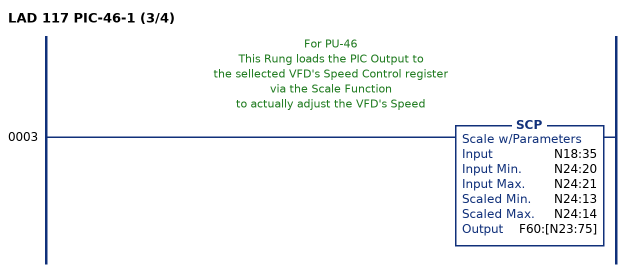
% Rung: 3 %
% For PU-46
% This Rung loads the PIC Output to
% the sellected VFD's Speed Control register
% via the Scale Function
% to actually adjust the VFD's Speed %
SOR SCP N18:35 N24:20 N24:21 N24:13 N24:14 F60:[N23:75] EOR
%   N18:35  PIC461_OUT1  "PIC-46-1 Flash Evap Feed Pres PID Output Value" %
%   N24:20  PID_MIN  "PID Statement Minimum Value" %
%   N24:21  PID_MAX  "PID Statement Maximum Value" %
%   N24:13  AO_MIN_OE4  "Analog Output Minimum Value Generates 4 mA DC (To OE4 AO Module)" %
%   N24:14  AO_MAX_OE4  "Analog Output Maximum Value Generates 20 mA DC (To OE4 AO Module)" %
%   N23:75  PIC461_OUT_PTR  "PIC-46-1 Flash Evap Feed Pres Output Pointer Determines which VFD is controled by FIC" %

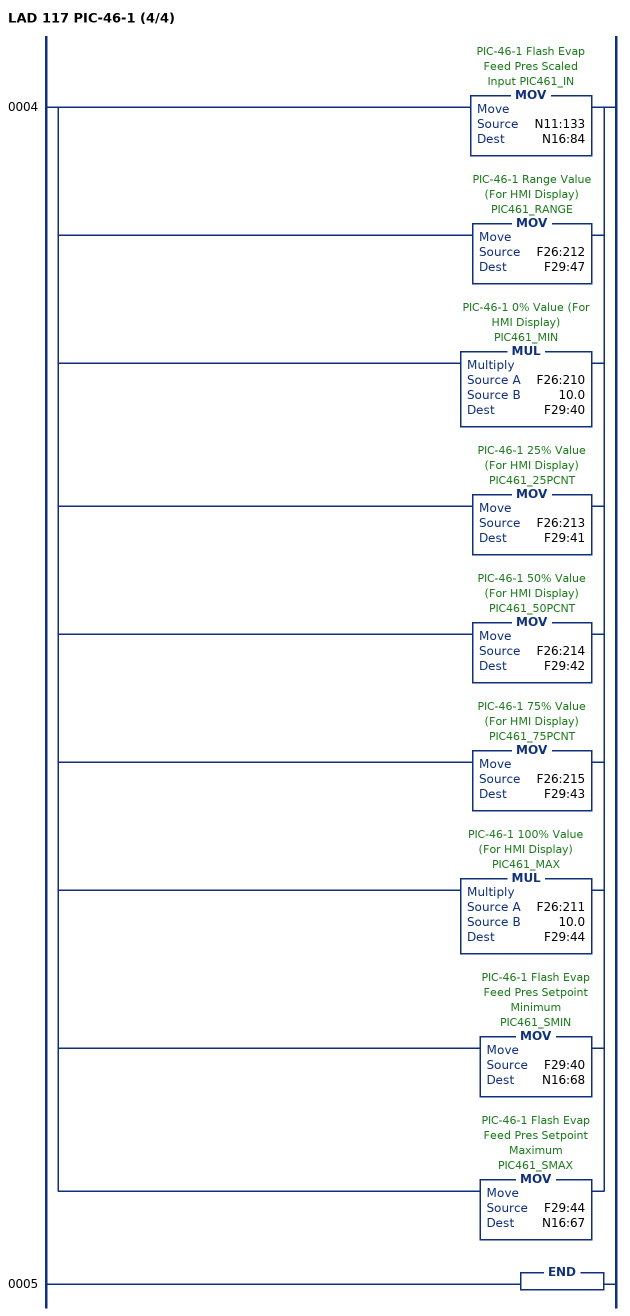
% Rung: 4 %
SOR BST MOV N11:133 N16:84 NXB MOV F26:212 F29:47 NXB MUL F26:210 10.0 F29:40 NXB MOV F26:213 F29:41 NXB MOV F26:214 F29:42 NXB MOV F26:215 F29:43 NXB MUL F26:211 10.0 F29:44 NXB MOV F29:40 N16:68 NXB MOV F29:44 N16:67 BND EOR
%   N11:133  PT461_PID_IN  "PT-46-1 Flash Evap Feed Pres PID Statement Input Value" %
%   N16:84  PIC461_IN  "PIC-46-1 Flash Evap Feed Pres Scaled Input" %
%   F26:212  PT461_RANGE  "PT-46-1 Range Value #NAME?" %
%   F29:47  PIC461_RANGE  "PIC-46-1 Range Value (For HMI Display)" %
%   F26:210  PT461_MIN  "PT-46-1 Minimum Value" %
%   F29:40  PIC461_MIN  "PIC-46-1 0% Value (For HMI Display)" %
%   F26:213  PT461_25PCNT_VALUE  "PT-46-1 25% Range Value For HMI Display" %
%   F29:41  PIC461_25PCNT  "PIC-46-1 25% Value (For HMI Display)" %
%   F26:214  PT461_50PCNT_VALUE  "PT-46-1 50% Range Value For HMI Display" %
%   F29:42  PIC461_50PCNT  "PIC-46-1 50% Value (For HMI Display)" %
%   F26:215  PT461_75PCNT_VALUE  "PT-46-1 75% Range Value For HMI Display" %
%   F29:43  PIC461_75PCNT  "PIC-46-1 75% Value (For HMI Display)" %
%   F26:211  PT461_MAX  "PT-46-1 Maximum Value" %
%   F29:44  PIC461_MAX  "PIC-46-1 100% Value (For HMI Display)" %
%   N16:68  PIC461_SMIN  "PIC-46-1 Flash Evap Feed Pres Setpoint Minimum" %
%   N16:67  PIC461_SMAX  "PIC-46-1 Flash Evap Feed Pres Setpoint Maximum" %
% Rung: 5 %
SOR END EOR

LADDER 121 "TIC-11-1"    % Tempered Water Loop No-1 Temperature PID Controls %
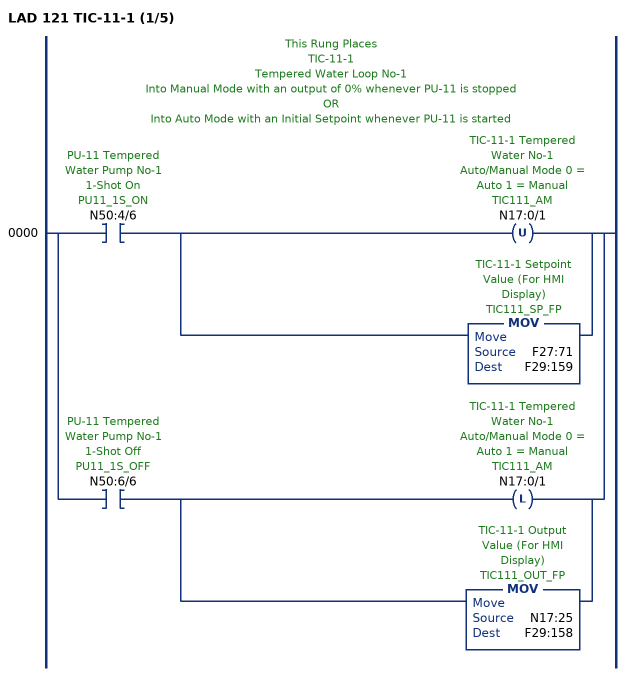
% Rung: 0 %
% This Rung Places
% TIC-11-1
% Tempered Water Loop No-1
% Into Manual Mode with an output of 0% whenever PU-11 is stopped
% OR
% Into Auto Mode with an Initial Setpoint whenever PU-11 is started %
SOR BST XIC N50:4/6 BST OTU N17:0/1 NXB MOV F27:71 F29:159 BND NXB XIC N50:6/6 BST OTL N17:0/1 NXB MOV N17:25 F29:158 BND BND EOR
%   N50:4/6  PU11_1S_ON  "PU-11 Tempered Water Pump No-1 1-Shot On" %
%   N17:0/1  TIC111_AM  "TIC-11-1 Tempered Water No-1 Auto/Manual Mode 0 = Auto 1 = Manual" %
%   F27:71  TIC111_INIT_SP  "TIC-11-1 Initial Temperature Setpoint" %
%   F29:159  TIC111_SP_FP  "TIC-11-1 Setpoint Value (For HMI Display)" %
%   N50:6/6  PU11_1S_OFF  "PU-11 Tempered Water Pump No-1 1-Shot Off" %
%   N17:25  TIC111_OFF_OUTPUT  "TIC-11-1 Output When PU-11 Is Off" %
%   F29:158  TIC111_OUT_FP  "TIC-11-1 Output Value (For HMI Display)" %

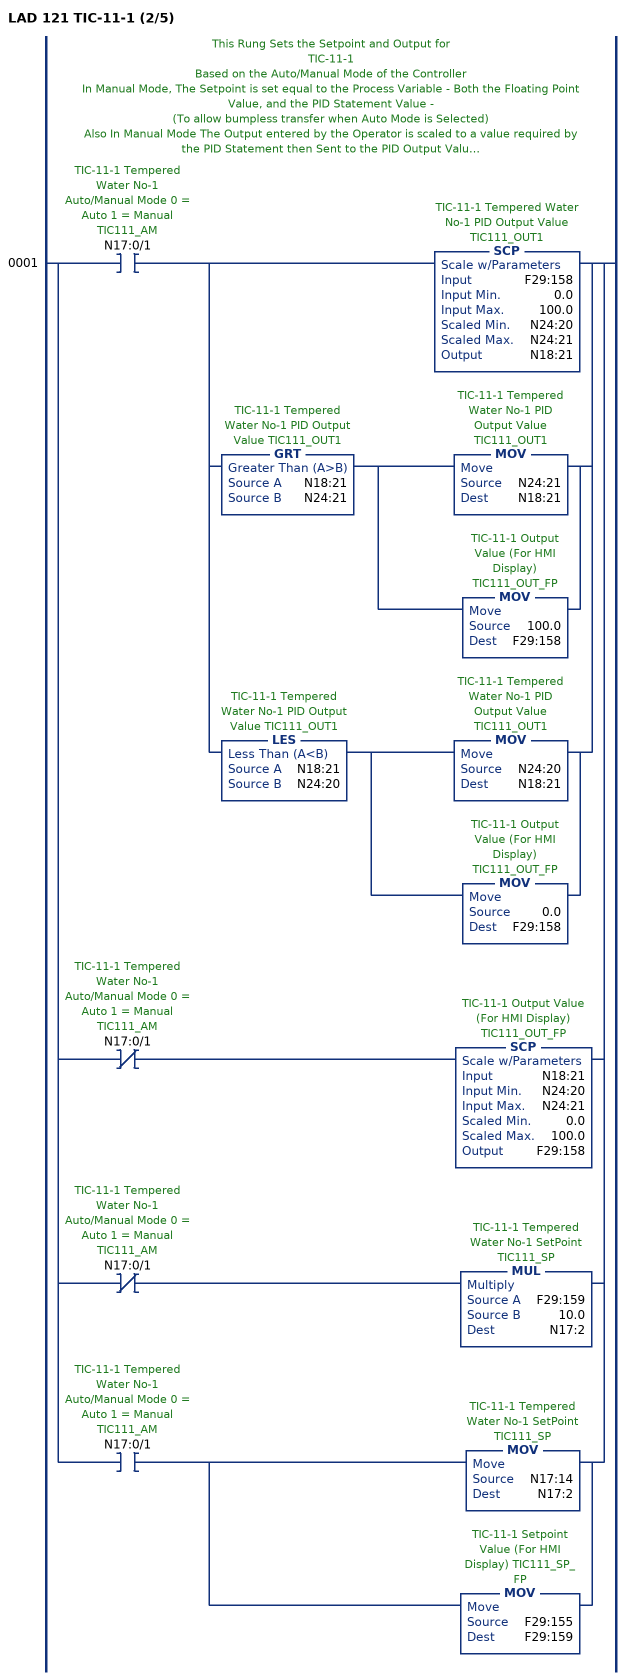
% Rung: 1 %
% This Rung Sets the Setpoint and Output for
% TIC-11-1
% Based on the Auto/Manual Mode of the Controller
% In Manual Mode, The Setpoint is set equal to the Process Variable - Both the Floating Point Value, and the PID Statement Value -
% (To allow bumpless transfer when Auto Mode is Selected)
% Also In Manual Mode The Output entered by the Operator is scaled to a value required by the PID Statement then Sent to the PID Output Value
% 
% In Auto Mode, The Setpoint is Entered by the Operator from Any HMI terminal, Multiplied by 10, and placed in the PID Statement's Setpoint Location
% Also In Auto Mode, the Output (used by the Operator) is set equal to the actual value of the pID statement
% (To allow bumpless transfer when Manual Mode is Selected) %
SOR BST XIC N17:0/1 BST SCP F29:158 0.0 100.0 N24:20 N24:21 N18:21 NXB GRT N18:21 N24:21 BST MOV N24:21 N18:21 NXB MOV 100.0 F29:158 BND NXB LES N18:21 N24:20 BST MOV N24:20 N18:21 NXB MOV 0.0 F29:158 BND BND NXB XIO N17:0/1 SCP N18:21 N24:20 N24:21 0.0 100.0 F29:158 NXB XIO N17:0/1 MUL F29:159 10.0 N17:2 NXB XIC N17:0/1 BST MOV N17:14 N17:2 NXB MOV F29:155 F29:159 BND BND EOR
%   N17:0/1  TIC111_AM  "TIC-11-1 Tempered Water No-1 Auto/Manual Mode 0 = Auto 1 = Manual" %
%   F29:158  TIC111_OUT_FP  "TIC-11-1 Output Value (For HMI Display)" %
%   N24:20  PID_MIN  "PID Statement Minimum Value" %
%   N24:21  PID_MAX  "PID Statement Maximum Value" %
%   N18:21  TIC111_OUT1  "TIC-11-1 Tempered Water No-1 PID Output Value" %
%   F29:159  TIC111_SP_FP  "TIC-11-1 Setpoint Value (For HMI Display)" %
%   N17:2  TIC111_SP  "TIC-11-1 Tempered Water No-1 SetPoint" %
%   N17:14  TIC111_PV  "TIC-11-1 Tempered Water No-1 Scaled Process Variable" %
%   F29:155  TIC111_PV_FP  "TIC-11-1 PV Value (For HMI Display)" %

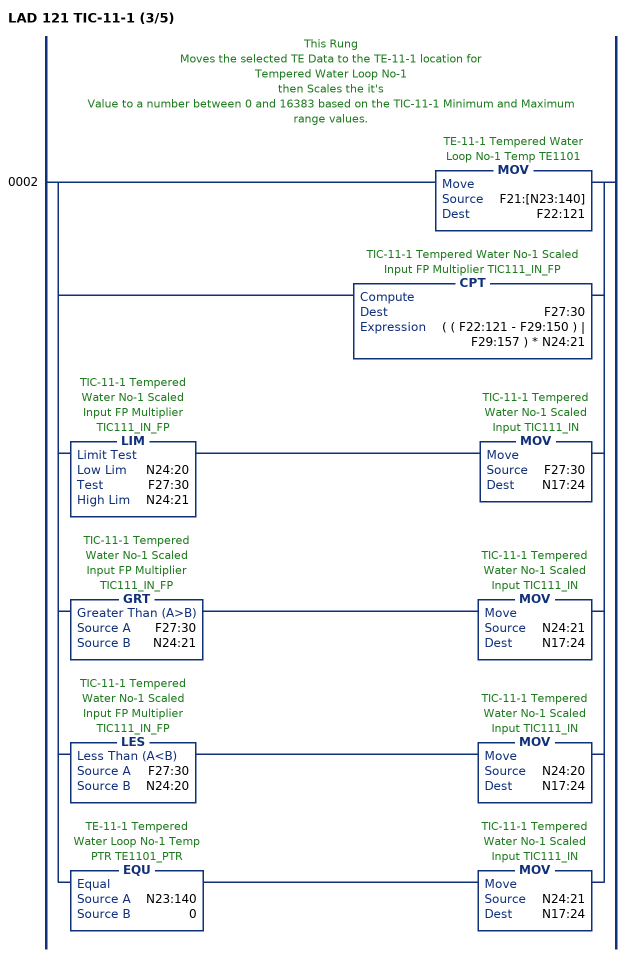
% Rung: 2 %
% This Rung
% Moves the selected TE Data to the TE-11-1 location for
% Tempered Water Loop No-1
% then Scales the it's
% Value to a number between 0 and 16383 based on the TIC-11-1 Minimum and Maximum range values. %
SOR BST MOV F21:[N23:140] F22:121 NXB CPT F27:30 " ( ( F22:121 - F29:150 ) | F29:157 ) * N24:21 " NXB LIM N24:20 F27:30 N24:21 MOV F27:30 N17:24 NXB GRT F27:30 N24:21 MOV N24:21 N17:24 NXB LES F27:30 N24:20 MOV N24:20 N17:24 NXB EQU N23:140 0 MOV N24:21 N17:24 BND EOR
%   N23:140  TE1101_PTR  "TE-11-1 Tempered Water Loop No-1 Temp PTR" %
%   F22:121  TE1101  "TE-11-1 Tempered Water Loop No-1 Temp" %
%   F27:30  TIC111_IN_FP  "TIC-11-1 Tempered Water No-1 Scaled Input FP Multiplier" %
%   F29:150  TIC111_MIN  "TIC-11-1 0% Value (For HMI Display)" %
%   F29:157  TIC111_RANGE  "TIC-11-1 Range Value (For HMI Display)" %
%   N24:21  PID_MAX  "PID Statement Maximum Value" %
%   N24:20  PID_MIN  "PID Statement Minimum Value" %
%   N17:24  TIC111_IN  "TIC-11-1 Tempered Water No-1 Scaled Input" %

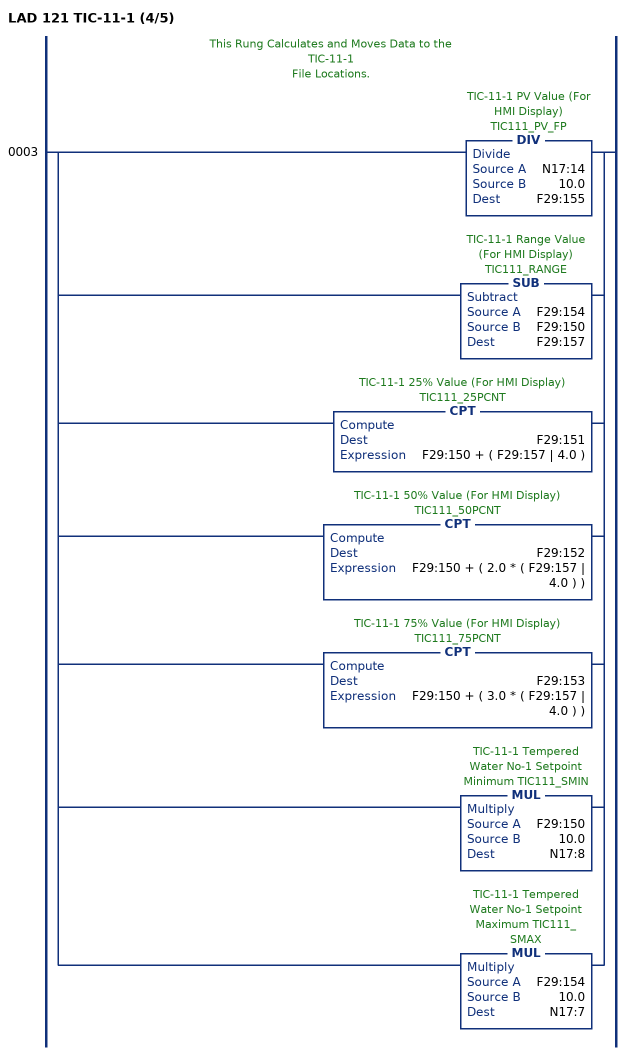
% Rung: 3 %
% This Rung Calculates and Moves Data to the
% TIC-11-1
% File Locations. %
SOR BST DIV N17:14 10.0 F29:155 NXB SUB F29:154 F29:150 F29:157 NXB CPT F29:151 " F29:150 + ( F29:157 | 4.0 ) " NXB CPT F29:152 " F29:150 + ( 2.0 * ( F29:157 | 4.0 ) ) " NXB CPT F29:153 " F29:150 + ( 3.0 * ( F29:157 | 4.0 ) ) " NXB MUL F29:150 10.0 N17:8 NXB MUL F29:154 10.0 N17:7 BND EOR
%   N17:14  TIC111_PV  "TIC-11-1 Tempered Water No-1 Scaled Process Variable" %
%   F29:155  TIC111_PV_FP  "TIC-11-1 PV Value (For HMI Display)" %
%   F29:154  TIC111_MAX  "TIC-11-1 100% Value (For HMI Display)" %
%   F29:150  TIC111_MIN  "TIC-11-1 0% Value (For HMI Display)" %
%   F29:157  TIC111_RANGE  "TIC-11-1 Range Value (For HMI Display)" %
%   F29:151  TIC111_25PCNT  "TIC-11-1 25% Value (For HMI Display)" %
%   F29:152  TIC111_50PCNT  "TIC-11-1 50% Value (For HMI Display)" %
%   F29:153  TIC111_75PCNT  "TIC-11-1 75% Value (For HMI Display)" %
%   N17:8  TIC111_SMIN  "TIC-11-1 Tempered Water No-1 Setpoint Minimum" %
%   N17:7  TIC111_SMAX  "TIC-11-1 Tempered Water No-1 Setpoint Maximum" %

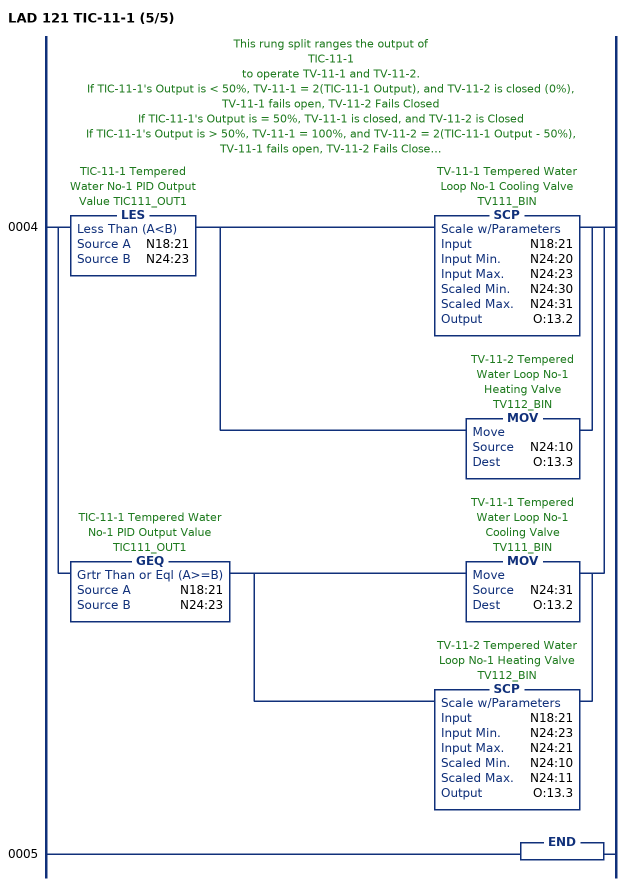
% Rung: 4 %
% This rung split ranges the output of
% TIC-11-1
% to operate TV-11-1 and TV-11-2.
% If TIC-11-1's Output is < 50%, TV-11-1 = 2(TIC-11-1 Output), and TV-11-2 is closed (0%), TV-11-1 fails open, TV-11-2 Fails Closed
% If TIC-11-1's Output is = 50%, TV-11-1 is closed, and TV-11-2 is Closed
% If TIC-11-1's Output is > 50%, TV-11-1 = 100%, and TV-11-2 = 2(TIC-11-1 Output - 50%), TV-11-1 fails open, TV-11-2 Fails Closed
% 
% TV-11-1 is 100% Open at ~0% Output, and Closed at 50% (TV-11-1 has problem, is Open at ~5madc and closed at ~ 12madc - This has been compensated for by modifing its SCALE function output values)
% TV-11-2 is Closed below 50% and Open at 100% %
SOR BST LES N18:21 N24:23 BST SCP N18:21 N24:20 N24:23 N24:30 N24:31 O:13.2 NXB MOV N24:10 O:13.3 BND NXB GEQ N18:21 N24:23 BST MOV N24:31 O:13.2 NXB SCP N18:21 N24:23 N24:21 N24:10 N24:11 O:13.3 BND BND EOR
%   N18:21  TIC111_OUT1  "TIC-11-1 Tempered Water No-1 PID Output Value" %
%   N24:23  PID_MID  "PID Statement Mid Value" %
%   N24:20  PID_MIN  "PID Statement Minimum Value" %
%   N24:30  TV111_AO_AT_OPEN  "TV-11-1 Loop 1 Cooling TV Analog Output at Open Position (~10% Signal)" %
%   N24:31  TV111_AO_AT_CLOSED  "TV-11-1 Loop 1 Cooling TV Analog Output at Closed Position (~50% Signal)" %
%   O:13.2  TV111_BIN  "TV-11-1 Tempered Water Loop No-1 Cooling Valve" %
%   N24:10  AO_MIN_NO4I  "Analog Output Minimum Value Generates 4 mA DC (To NO4I AO Module)" %
%   O:13.3  TV112_BIN  "TV-11-2 Tempered Water Loop No-1 Heating Valve" %
%   N24:21  PID_MAX  "PID Statement Maximum Value" %
%   N24:11  AO_MAX_NO4I  "Analog Output Maximum Value Generates 20 mA DC (To NO4I AO Module)" %
% Rung: 5 %
SOR END EOR

LADDER 122 "TIC-12-1"    % Tempered Water Loop No-2 Temperature PID Controls %
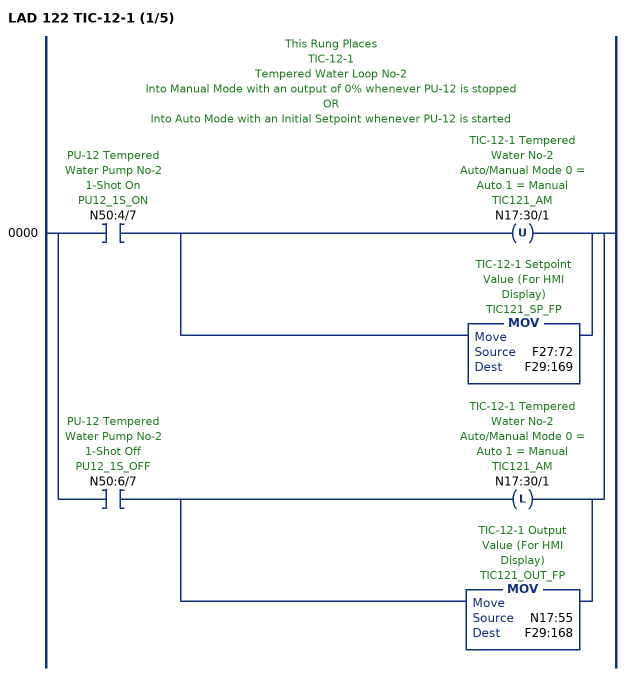
% Rung: 0 %
% This Rung Places
% TIC-12-1
% Tempered Water Loop No-2
% Into Manual Mode with an output of 0% whenever PU-12 is stopped
% OR
% Into Auto Mode with an Initial Setpoint whenever PU-12 is started %
SOR BST XIC N50:4/7 BST OTU N17:30/1 NXB MOV F27:72 F29:169 BND NXB XIC N50:6/7 BST OTL N17:30/1 NXB MOV N17:55 F29:168 BND BND EOR
%   N50:4/7  PU12_1S_ON  "PU-12 Tempered Water Pump No-2 1-Shot On" %
%   N17:30/1  TIC121_AM  "TIC-12-1 Tempered Water No-2 Auto/Manual Mode 0 = Auto 1 = Manual" %
%   F27:72  TIC121_INIT_SP  "TIC-12-1 Initial Temperature Setpoint" %
%   F29:169  TIC121_SP_FP  "TIC-12-1 Setpoint Value (For HMI Display)" %
%   N50:6/7  PU12_1S_OFF  "PU-12 Tempered Water Pump No-2 1-Shot Off" %
%   N17:55  TIC121_OFF_OUTPUT  "TIC-12-1 Output When PU-12 Is Off" %
%   F29:168  TIC121_OUT_FP  "TIC-12-1 Output Value (For HMI Display)" %

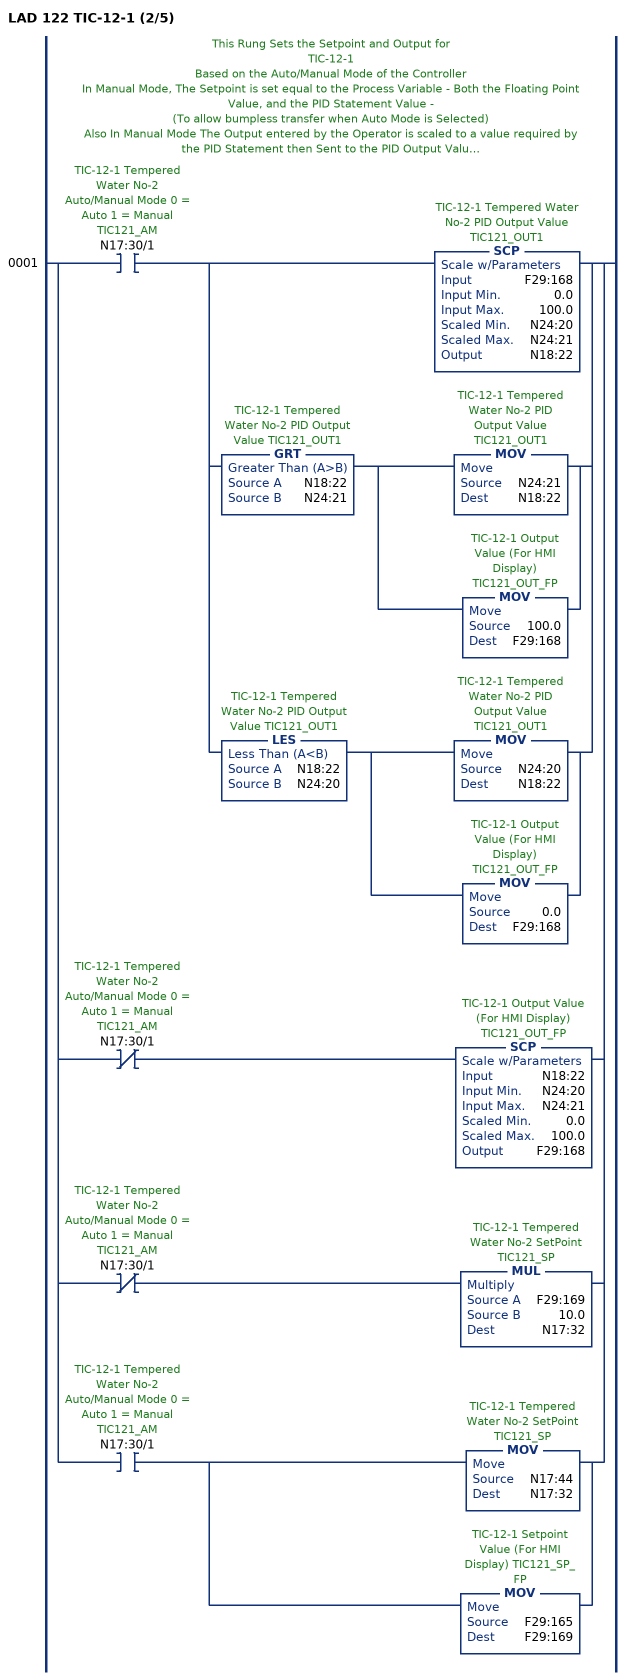
% Rung: 1 %
% This Rung Sets the Setpoint and Output for
% TIC-12-1
% Based on the Auto/Manual Mode of the Controller
% In Manual Mode, The Setpoint is set equal to the Process Variable - Both the Floating Point Value, and the PID Statement Value -
% (To allow bumpless transfer when Auto Mode is Selected)
% Also In Manual Mode The Output entered by the Operator is scaled to a value required by the PID Statement then Sent to the PID Output Value
% 
% In Auto Mode, The Setpoint is Entered by the Operator from Any HMI terminal, Multiplied by 10, and placed in the PID Statement's Setpoint Location
% Also In Auto Mode, the Output (used by the Operator) is set equal to the actual value of the pID statement
% (To allow bumpless transfer when Manual Mode is Selected) %
SOR BST XIC N17:30/1 BST SCP F29:168 0.0 100.0 N24:20 N24:21 N18:22 NXB GRT N18:22 N24:21 BST MOV N24:21 N18:22 NXB MOV 100.0 F29:168 BND NXB LES N18:22 N24:20 BST MOV N24:20 N18:22 NXB MOV 0.0 F29:168 BND BND NXB XIO N17:30/1 SCP N18:22 N24:20 N24:21 0.0 100.0 F29:168 NXB XIO N17:30/1 MUL F29:169 10.0 N17:32 NXB XIC N17:30/1 BST MOV N17:44 N17:32 NXB MOV F29:165 F29:169 BND BND EOR
%   N17:30/1  TIC121_AM  "TIC-12-1 Tempered Water No-2 Auto/Manual Mode 0 = Auto 1 = Manual" %
%   F29:168  TIC121_OUT_FP  "TIC-12-1 Output Value (For HMI Display)" %
%   N24:20  PID_MIN  "PID Statement Minimum Value" %
%   N24:21  PID_MAX  "PID Statement Maximum Value" %
%   N18:22  TIC121_OUT1  "TIC-12-1 Tempered Water No-2 PID Output Value" %
%   F29:169  TIC121_SP_FP  "TIC-12-1 Setpoint Value (For HMI Display)" %
%   N17:32  TIC121_SP  "TIC-12-1 Tempered Water No-2 SetPoint" %
%   N17:44  TIC121_PV  "TIC-12-1 Tempered Water No-2 Scaled Process Variable" %
%   F29:165  TIC121_PV_FP  "TIC-12-1 PV Value (For HMI Display)" %

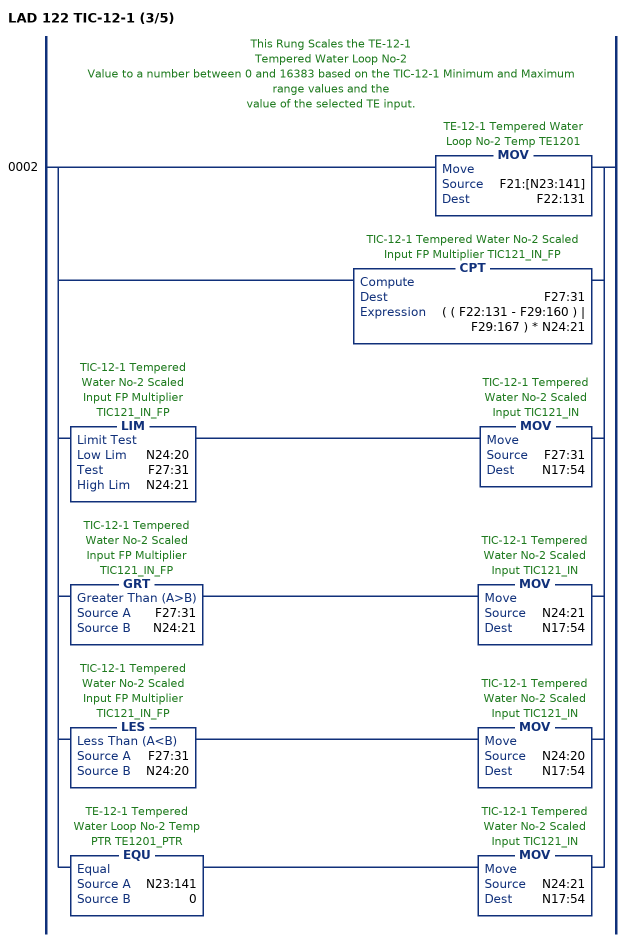
% Rung: 2 %
% This Rung Scales the TE-12-1
% Tempered Water Loop No-2
% Value to a number between 0 and 16383 based on the TIC-12-1 Minimum and Maximum range values and the
% value of the selected TE input. %
SOR BST MOV F21:[N23:141] F22:131 NXB CPT F27:31 " ( ( F22:131 - F29:160 ) | F29:167 ) * N24:21 " NXB LIM N24:20 F27:31 N24:21 MOV F27:31 N17:54 NXB GRT F27:31 N24:21 MOV N24:21 N17:54 NXB LES F27:31 N24:20 MOV N24:20 N17:54 NXB EQU N23:141 0 MOV N24:21 N17:54 BND EOR
%   N23:141  TE1201_PTR  "TE-12-1 Tempered Water Loop No-2 Temp PTR" %
%   F22:131  TE1201  "TE-12-1 Tempered Water Loop No-2 Temp" %
%   F27:31  TIC121_IN_FP  "TIC-12-1 Tempered Water No-2 Scaled Input FP Multiplier" %
%   F29:160  TIC121_MIN  "TIC-12-1 0% Value (For HMI Display)" %
%   F29:167  TIC121_RANGE  "TIC-12-1 Range Value (For HMI Display)" %
%   N24:21  PID_MAX  "PID Statement Maximum Value" %
%   N24:20  PID_MIN  "PID Statement Minimum Value" %
%   N17:54  TIC121_IN  "TIC-12-1 Tempered Water No-2 Scaled Input" %

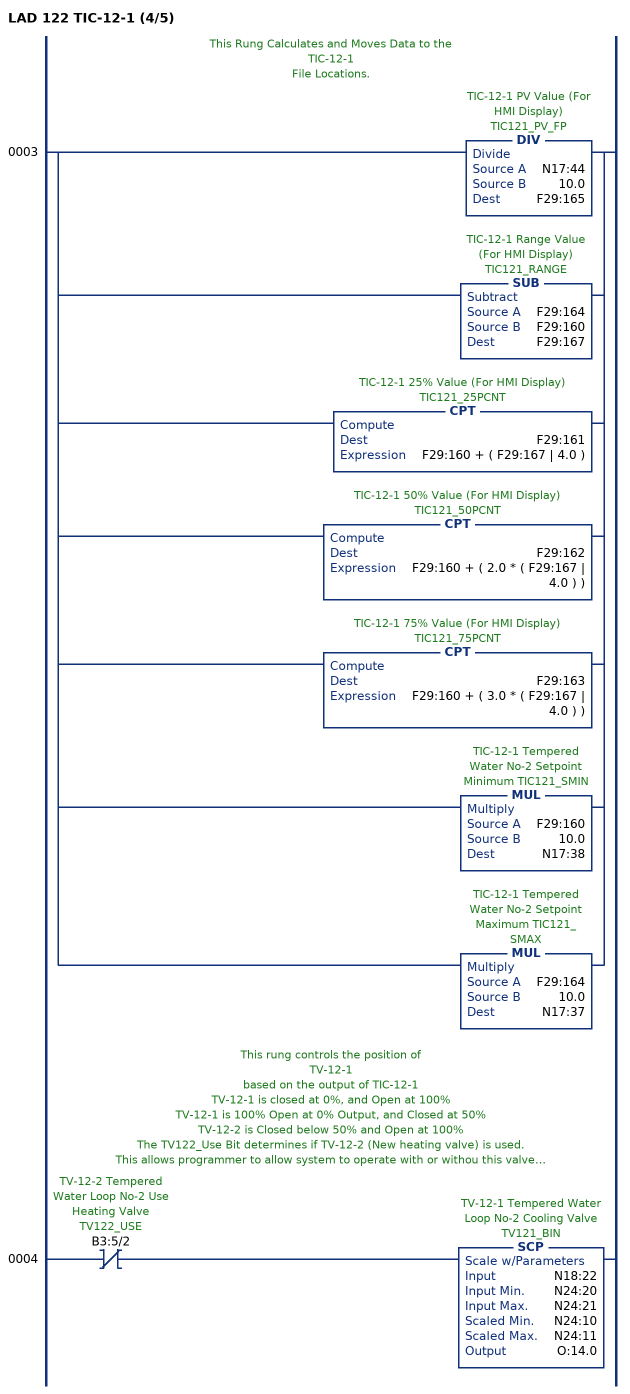
% Rung: 3 %
% This Rung Calculates and Moves Data to the
% TIC-12-1
% File Locations. %
SOR BST DIV N17:44 10.0 F29:165 NXB SUB F29:164 F29:160 F29:167 NXB CPT F29:161 " F29:160 + ( F29:167 | 4.0 ) " NXB CPT F29:162 " F29:160 + ( 2.0 * ( F29:167 | 4.0 ) ) " NXB CPT F29:163 " F29:160 + ( 3.0 * ( F29:167 | 4.0 ) ) " NXB MUL F29:160 10.0 N17:38 NXB MUL F29:164 10.0 N17:37 BND EOR
%   N17:44  TIC121_PV  "TIC-12-1 Tempered Water No-2 Scaled Process Variable" %
%   F29:165  TIC121_PV_FP  "TIC-12-1 PV Value (For HMI Display)" %
%   F29:164  TIC121_MAX  "TIC-12-1 100% Value (For HMI Display)" %
%   F29:160  TIC121_MIN  "TIC-12-1 0% Value (For HMI Display)" %
%   F29:167  TIC121_RANGE  "TIC-12-1 Range Value (For HMI Display)" %
%   F29:161  TIC121_25PCNT  "TIC-12-1 25% Value (For HMI Display)" %
%   F29:162  TIC121_50PCNT  "TIC-12-1 50% Value (For HMI Display)" %
%   F29:163  TIC121_75PCNT  "TIC-12-1 75% Value (For HMI Display)" %
%   N17:38  TIC121_SMIN  "TIC-12-1 Tempered Water No-2 Setpoint Minimum" %
%   N17:37  TIC121_SMAX  "TIC-12-1 Tempered Water No-2 Setpoint Maximum" %
% Rung: 4 %
% This rung controls the position of
% TV-12-1
% based on the output of TIC-12-1
% TV-12-1 is closed at 0%, and Open at 100%
% 
% TV-12-1 is 100% Open at 0% Output, and Closed at 50%
% TV-12-2 is Closed below 50% and Open at 100%
% 
% The TV122_Use Bit determines if TV-12-2 (New heating valve) is used.
% This allows programmer to allow system to operate with or withou this valve.
% Once the valve is permenantly install, this rung can be deleted %
SOR XIO B3:5/2 SCP N18:22 N24:20 N24:21 N24:10 N24:11 O:14.0 EOR
%   B3:5/2  TV122_USE  "TV-12-2 Tempered Water Loop No-2 Use Heating Valve" %
%   N18:22  TIC121_OUT1  "TIC-12-1 Tempered Water No-2 PID Output Value" %
%   N24:20  PID_MIN  "PID Statement Minimum Value" %
%   N24:21  PID_MAX  "PID Statement Maximum Value" %
%   N24:10  AO_MIN_NO4I  "Analog Output Minimum Value Generates 4 mA DC (To NO4I AO Module)" %
%   N24:11  AO_MAX_NO4I  "Analog Output Maximum Value Generates 20 mA DC (To NO4I AO Module)" %
%   O:14.0  TV121_BIN  "TV-12-1 Tempered Water Loop No-2 Cooling Valve" %

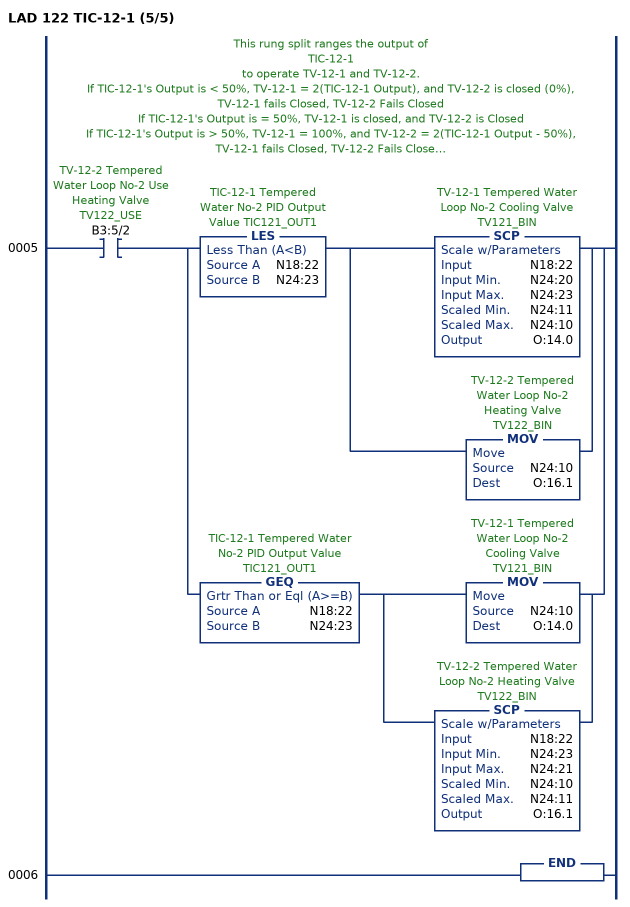
% Rung: 5 %
% This rung split ranges the output of
% TIC-12-1
% to operate TV-12-1 and TV-12-2.
% If TIC-12-1's Output is < 50%, TV-12-1 = 2(TIC-12-1 Output), and TV-12-2 is closed (0%), TV-12-1 fails Closed, TV-12-2 Fails Closed
% If TIC-12-1's Output is = 50%, TV-12-1 is closed, and TV-12-2 is Closed
% If TIC-12-1's Output is > 50%, TV-12-1 = 100%, and TV-12-2 = 2(TIC-12-1 Output - 50%), TV-12-1 fails Closed, TV-12-2 Fails Closed
% 
% TV-12-1 is 100% Open at 0% Output, and Closed at 50%
% TV-12-2 is Closed below 50% and Open at 100%
% 
% The TV122_Use Bit determines if TV-12-2 (New heating valve) is used.
% This allows programmer to allow system to operate with or withou this valve.
% Once the valve is permenantly install, the rung above this can be deleted and the contact removed on this rung %
SOR XIC B3:5/2 BST LES N18:22 N24:23 BST SCP N18:22 N24:20 N24:23 N24:11 N24:10 O:14.0 NXB MOV N24:10 O:16.1 BND NXB GEQ N18:22 N24:23 BST MOV N24:10 O:14.0 NXB SCP N18:22 N24:23 N24:21 N24:10 N24:11 O:16.1 BND BND EOR
%   B3:5/2  TV122_USE  "TV-12-2 Tempered Water Loop No-2 Use Heating Valve" %
%   N18:22  TIC121_OUT1  "TIC-12-1 Tempered Water No-2 PID Output Value" %
%   N24:23  PID_MID  "PID Statement Mid Value" %
%   N24:20  PID_MIN  "PID Statement Minimum Value" %
%   N24:11  AO_MAX_NO4I  "Analog Output Maximum Value Generates 20 mA DC (To NO4I AO Module)" %
%   N24:10  AO_MIN_NO4I  "Analog Output Minimum Value Generates 4 mA DC (To NO4I AO Module)" %
%   O:14.0  TV121_BIN  "TV-12-1 Tempered Water Loop No-2 Cooling Valve" %
%   O:16.1  TV122_BIN  "TV-12-2 Tempered Water Loop No-2 Heating Valve" %
%   N24:21  PID_MAX  "PID Statement Maximum Value" %
% Rung: 6 %
SOR END EOR

LADDER 123 "TIC-15-1"    % Tempered Oil Loop No-1 Temperature PID Controls %
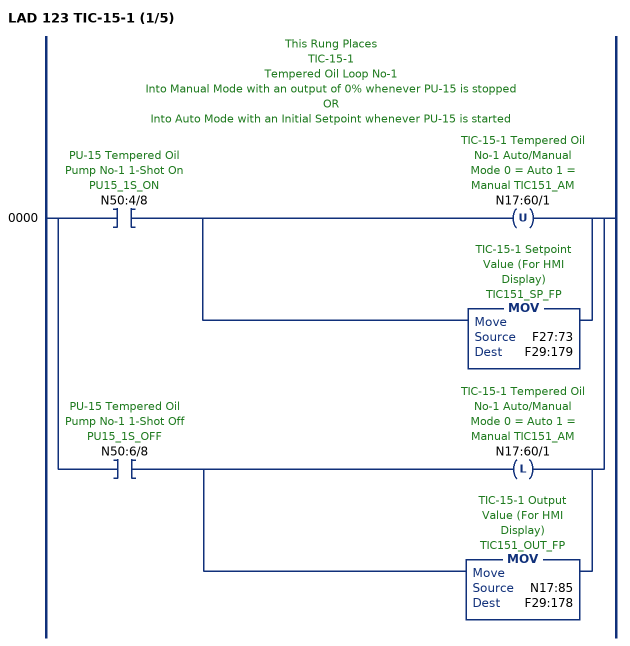
% Rung: 0 %
% This Rung Places
% TIC-15-1
% Tempered Oil Loop No-1
% Into Manual Mode with an output of 0% whenever PU-15 is stopped
% OR
% Into Auto Mode with an Initial Setpoint whenever PU-15 is started %
SOR BST XIC N50:4/8 BST OTU N17:60/1 NXB MOV F27:73 F29:179 BND NXB XIC N50:6/8 BST OTL N17:60/1 NXB MOV N17:85 F29:178 BND BND EOR
%   N50:4/8  PU15_1S_ON  "PU-15 Tempered Oil Pump No-1 1-Shot On" %
%   N17:60/1  TIC151_AM  "TIC-15-1 Tempered Oil No-1 Auto/Manual Mode 0 = Auto 1 = Manual" %
%   F27:73  TIC151_INIT_SP  "TIC-15-1 Initial Temperature Setpoint" %
%   F29:179  TIC151_SP_FP  "TIC-15-1 Setpoint Value (For HMI Display)" %
%   N50:6/8  PU15_1S_OFF  "PU-15 Tempered Oil Pump No-1 1-Shot Off" %
%   N17:85  TIC151_OFF_OUTPUT  "TIC-15-1 Output When PU-15 Is Off" %
%   F29:178  TIC151_OUT_FP  "TIC-15-1 Output Value (For HMI Display)" %

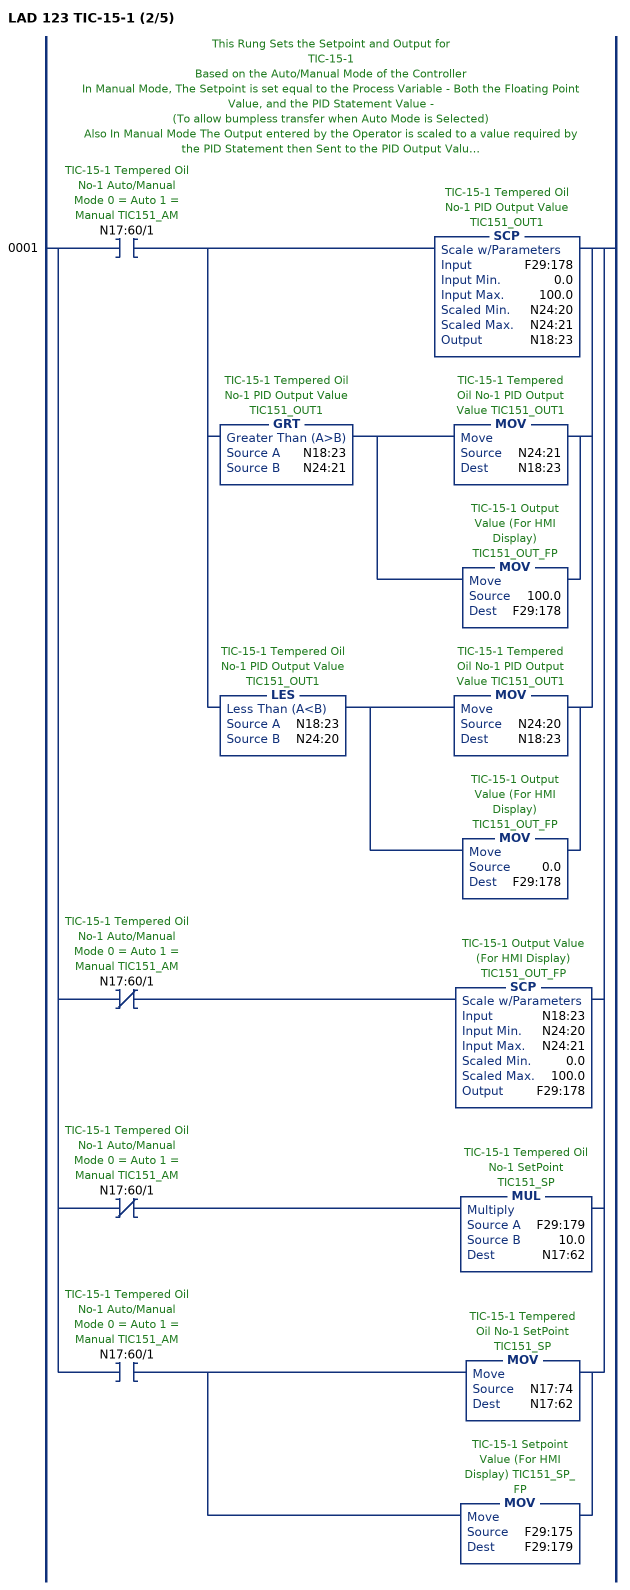
% Rung: 1 %
% This Rung Sets the Setpoint and Output for
% TIC-15-1
% Based on the Auto/Manual Mode of the Controller
% In Manual Mode, The Setpoint is set equal to the Process Variable - Both the Floating Point Value, and the PID Statement Value -
% (To allow bumpless transfer when Auto Mode is Selected)
% Also In Manual Mode The Output entered by the Operator is scaled to a value required by the PID Statement then Sent to the PID Output Value
% 
% In Auto Mode, The Setpoint is Entered by the Operator from Any HMI terminal, Multiplied by 10, and placed in the PID Statement's Setpoint Location
% Also In Auto Mode, the Output (used by the Operator) is set equal to the actual value of the pID statement
% (To allow bumpless transfer when Manual Mode is Selected) %
SOR BST XIC N17:60/1 BST SCP F29:178 0.0 100.0 N24:20 N24:21 N18:23 NXB GRT N18:23 N24:21 BST MOV N24:21 N18:23 NXB MOV 100.0 F29:178 BND NXB LES N18:23 N24:20 BST MOV N24:20 N18:23 NXB MOV 0.0 F29:178 BND BND NXB XIO N17:60/1 SCP N18:23 N24:20 N24:21 0.0 100.0 F29:178 NXB XIO N17:60/1 MUL F29:179 10.0 N17:62 NXB XIC N17:60/1 BST MOV N17:74 N17:62 NXB MOV F29:175 F29:179 BND BND EOR
%   N17:60/1  TIC151_AM  "TIC-15-1 Tempered Oil No-1 Auto/Manual Mode 0 = Auto 1 = Manual" %
%   F29:178  TIC151_OUT_FP  "TIC-15-1 Output Value (For HMI Display)" %
%   N24:20  PID_MIN  "PID Statement Minimum Value" %
%   N24:21  PID_MAX  "PID Statement Maximum Value" %
%   N18:23  TIC151_OUT1  "TIC-15-1 Tempered Oil No-1 PID Output Value" %
%   F29:179  TIC151_SP_FP  "TIC-15-1 Setpoint Value (For HMI Display)" %
%   N17:62  TIC151_SP  "TIC-15-1 Tempered Oil No-1 SetPoint" %
%   N17:74  TIC151_PV  "TIC-15-1 Tempered Oil No-1 Scaled Process Variable" %
%   F29:175  TIC151_PV_FP  "TIC-15-1 PV Value (For HMI Display)" %

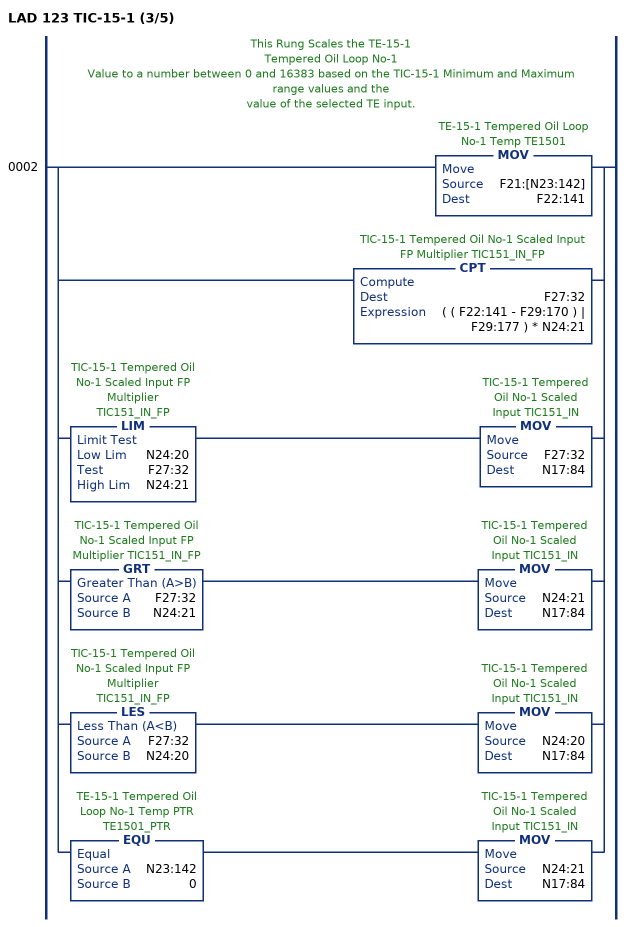
% Rung: 2 %
% This Rung Scales the TE-15-1
% Tempered Oil Loop No-1
% Value to a number between 0 and 16383 based on the TIC-15-1 Minimum and Maximum range values and the
% value of the selected TE input. %
SOR BST MOV F21:[N23:142] F22:141 NXB CPT F27:32 " ( ( F22:141 - F29:170 ) | F29:177 ) * N24:21 " NXB LIM N24:20 F27:32 N24:21 MOV F27:32 N17:84 NXB GRT F27:32 N24:21 MOV N24:21 N17:84 NXB LES F27:32 N24:20 MOV N24:20 N17:84 NXB EQU N23:142 0 MOV N24:21 N17:84 BND EOR
%   N23:142  TE1501_PTR  "TE-15-1 Tempered Oil Loop No-1 Temp PTR" %
%   F22:141  TE1501  "TE-15-1 Tempered Oil Loop No-1 Temp" %
%   F27:32  TIC151_IN_FP  "TIC-15-1 Tempered Oil No-1 Scaled Input FP Multiplier" %
%   F29:170  TIC151_MIN  "TIC-15-1 0% Value (For HMI Display)" %
%   F29:177  TIC151_RANGE  "TIC-15-1 Range Value (For HMI Display)" %
%   N24:21  PID_MAX  "PID Statement Maximum Value" %
%   N24:20  PID_MIN  "PID Statement Minimum Value" %
%   N17:84  TIC151_IN  "TIC-15-1 Tempered Oil No-1 Scaled Input" %

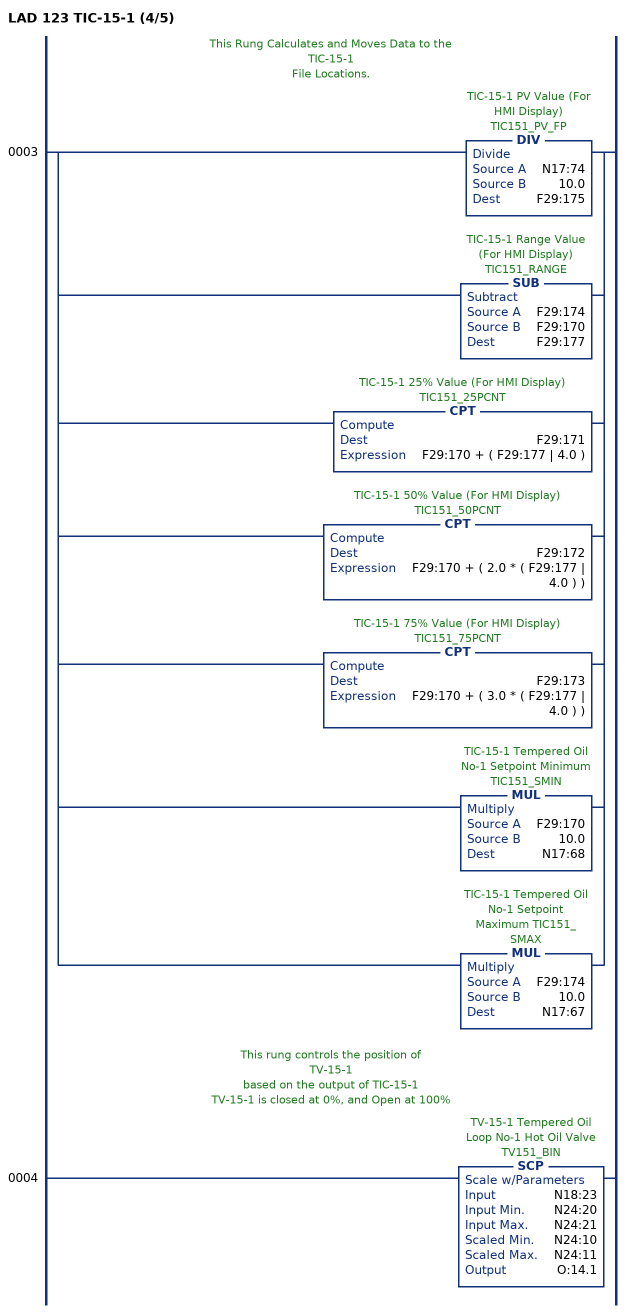
% Rung: 3 %
% This Rung Calculates and Moves Data to the
% TIC-15-1
% File Locations. %
SOR BST DIV N17:74 10.0 F29:175 NXB SUB F29:174 F29:170 F29:177 NXB CPT F29:171 " F29:170 + ( F29:177 | 4.0 ) " NXB CPT F29:172 " F29:170 + ( 2.0 * ( F29:177 | 4.0 ) ) " NXB CPT F29:173 " F29:170 + ( 3.0 * ( F29:177 | 4.0 ) ) " NXB MUL F29:170 10.0 N17:68 NXB MUL F29:174 10.0 N17:67 BND EOR
%   N17:74  TIC151_PV  "TIC-15-1 Tempered Oil No-1 Scaled Process Variable" %
%   F29:175  TIC151_PV_FP  "TIC-15-1 PV Value (For HMI Display)" %
%   F29:174  TIC151_MAX  "TIC-15-1 100% Value (For HMI Display)" %
%   F29:170  TIC151_MIN  "TIC-15-1 0% Value (For HMI Display)" %
%   F29:177  TIC151_RANGE  "TIC-15-1 Range Value (For HMI Display)" %
%   F29:171  TIC151_25PCNT  "TIC-15-1 25% Value (For HMI Display)" %
%   F29:172  TIC151_50PCNT  "TIC-15-1 50% Value (For HMI Display)" %
%   F29:173  TIC151_75PCNT  "TIC-15-1 75% Value (For HMI Display)" %
%   N17:68  TIC151_SMIN  "TIC-15-1 Tempered Oil No-1 Setpoint Minimum" %
%   N17:67  TIC151_SMAX  "TIC-15-1 Tempered Oil No-1 Setpoint Maximum" %
% Rung: 4 %
% This rung controls the position of
% TV-15-1
% based on the output of TIC-15-1
% TV-15-1 is closed at 0%, and Open at 100% %
SOR SCP N18:23 N24:20 N24:21 N24:10 N24:11 O:14.1 EOR
%   N18:23  TIC151_OUT1  "TIC-15-1 Tempered Oil No-1 PID Output Value" %
%   N24:20  PID_MIN  "PID Statement Minimum Value" %
%   N24:21  PID_MAX  "PID Statement Maximum Value" %
%   N24:10  AO_MIN_NO4I  "Analog Output Minimum Value Generates 4 mA DC (To NO4I AO Module)" %
%   N24:11  AO_MAX_NO4I  "Analog Output Maximum Value Generates 20 mA DC (To NO4I AO Module)" %
%   O:14.1  TV151_BIN  "TV-15-1 Tempered Oil Loop No-1 Hot Oil Valve" %

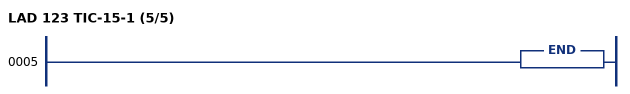
% Rung: 5 %
SOR END EOR

LADDER 124 "TIC-24-1"    % Hot Oil Temperature PID Controls %
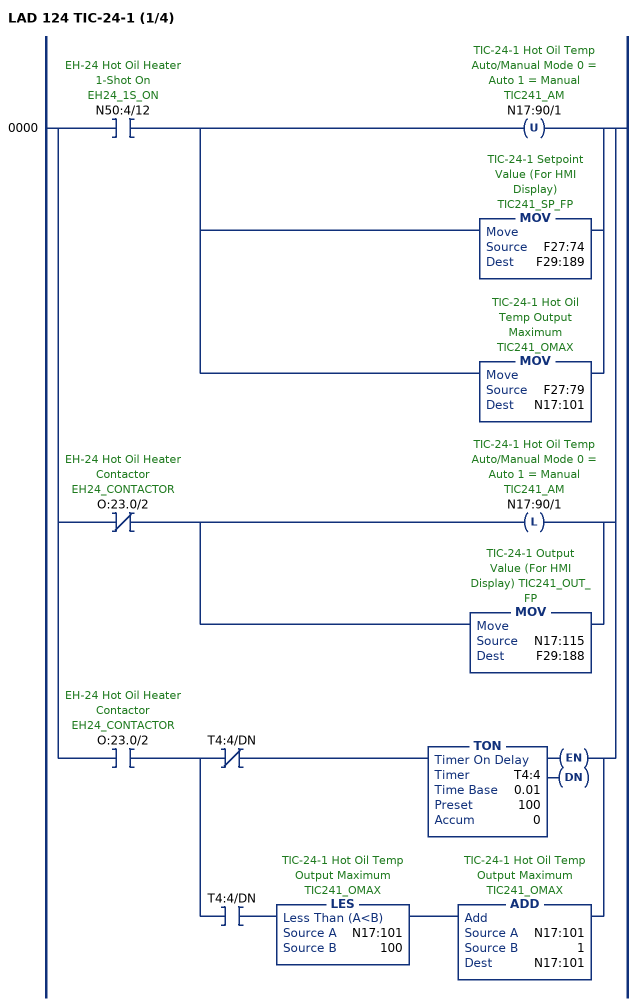
% Rung: 0 %
SOR BST XIC N50:4/12 BST OTU N17:90/1 NXB MOV F27:74 F29:189 NXB MOV F27:79 N17:101 BND NXB XIO O:23.0/2 BST OTL N17:90/1 NXB MOV N17:115 F29:188 BND NXB XIC O:23.0/2 BST XIO T4:4/DN TON T4:4 0.01 100 0 NXB XIC T4:4/DN LES N17:101 100 ADD N17:101 1 N17:101 BND BND EOR
%   N50:4/12  EH24_1S_ON  "EH-24 Hot Oil Heater 1-Shot On" %
%   N17:90/1  TIC241_AM  "TIC-24-1 Hot Oil Temp Auto/Manual Mode 0 = Auto 1 = Manual" %
%   F27:74  TIC241_INIT_SP  "TIC-24-1 Initial Temperature Setpoint" %
%   F29:189  TIC241_SP_FP  "TIC-24-1 Setpoint Value (For HMI Display)" %
%   F27:79  TIC241_INIT_OUTPUT  "TIC-24-1 Initial Output" %
%   N17:101  TIC241_OMAX  "TIC-24-1 Hot Oil Temp Output Maximum" %
%   O:23.0/2  EH24_CONTACTOR  "EH-24 Hot Oil Heater Contactor" %
%   N17:115  TIC241_OFF_OUTPUT  "TIC-24-1 Output When PU-23 Is Off" %
%   F29:188  TIC241_OUT_FP  "TIC-24-1 Output Value (For HMI Display)" %

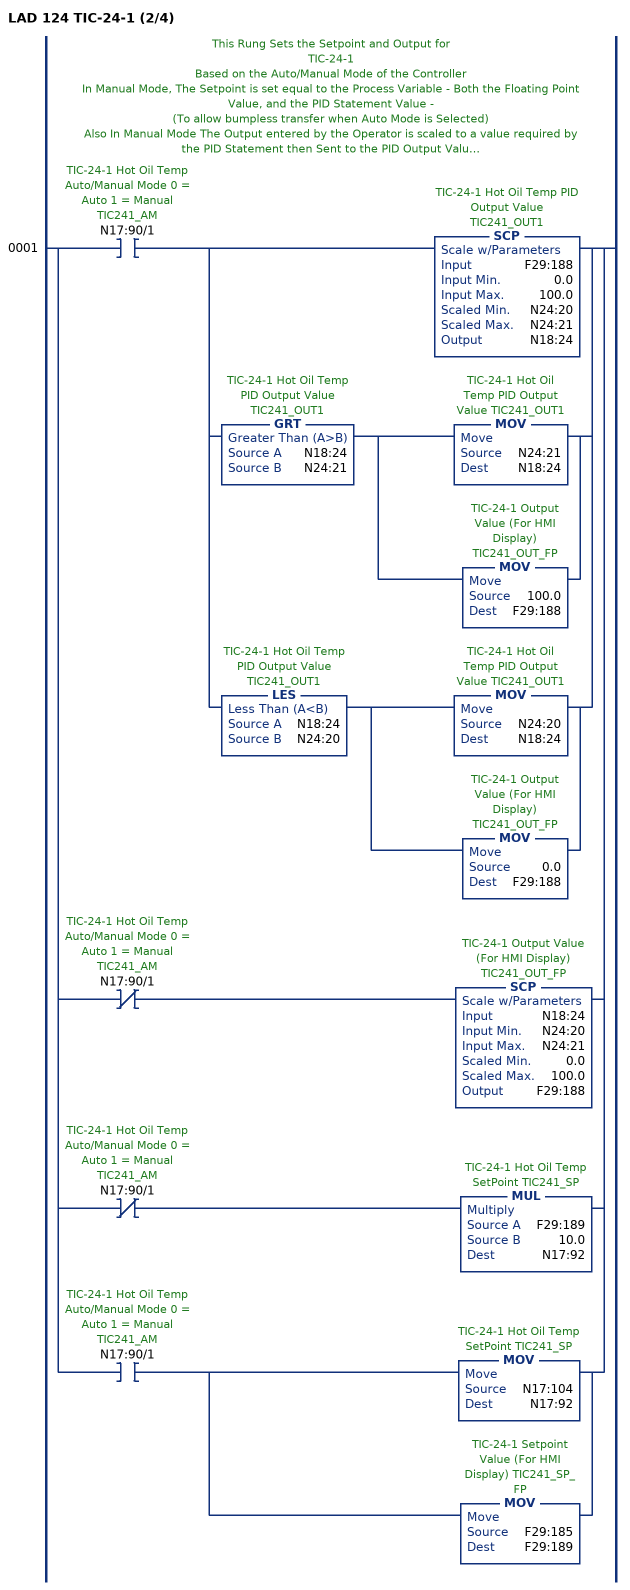
% Rung: 1 %
% This Rung Sets the Setpoint and Output for
% TIC-24-1
% Based on the Auto/Manual Mode of the Controller
% In Manual Mode, The Setpoint is set equal to the Process Variable - Both the Floating Point Value, and the PID Statement Value -
% (To allow bumpless transfer when Auto Mode is Selected)
% Also In Manual Mode The Output entered by the Operator is scaled to a value required by the PID Statement then Sent to the PID Output Value
% 
% In Auto Mode, The Setpoint is Entered by the Operator from Any HMI terminal, Multiplied by 10, and placed in the PID Statement's Setpoint Location
% Also In Auto Mode, the Output (used by the Operator) is set equal to the actual value of the pID statement
% (To allow bumpless transfer when Manual Mode is Selected) %
SOR BST XIC N17:90/1 BST SCP F29:188 0.0 100.0 N24:20 N24:21 N18:24 NXB GRT N18:24 N24:21 BST MOV N24:21 N18:24 NXB MOV 100.0 F29:188 BND NXB LES N18:24 N24:20 BST MOV N24:20 N18:24 NXB MOV 0.0 F29:188 BND BND NXB XIO N17:90/1 SCP N18:24 N24:20 N24:21 0.0 100.0 F29:188 NXB XIO N17:90/1 MUL F29:189 10.0 N17:92 NXB XIC N17:90/1 BST MOV N17:104 N17:92 NXB MOV F29:185 F29:189 BND BND EOR
%   N17:90/1  TIC241_AM  "TIC-24-1 Hot Oil Temp Auto/Manual Mode 0 = Auto 1 = Manual" %
%   F29:188  TIC241_OUT_FP  "TIC-24-1 Output Value (For HMI Display)" %
%   N24:20  PID_MIN  "PID Statement Minimum Value" %
%   N24:21  PID_MAX  "PID Statement Maximum Value" %
%   N18:24  TIC241_OUT1  "TIC-24-1 Hot Oil Temp PID Output Value" %
%   F29:189  TIC241_SP_FP  "TIC-24-1 Setpoint Value (For HMI Display)" %
%   N17:92  TIC241_SP  "TIC-24-1 Hot Oil Temp SetPoint" %
%   N17:104  TIC241_PV  "TIC-24-1 Hot Oil Temp Scaled Process Variable" %
%   F29:185  TIC241_PV_FP  "TIC-24-1 PV Value (For HMI Display)" %

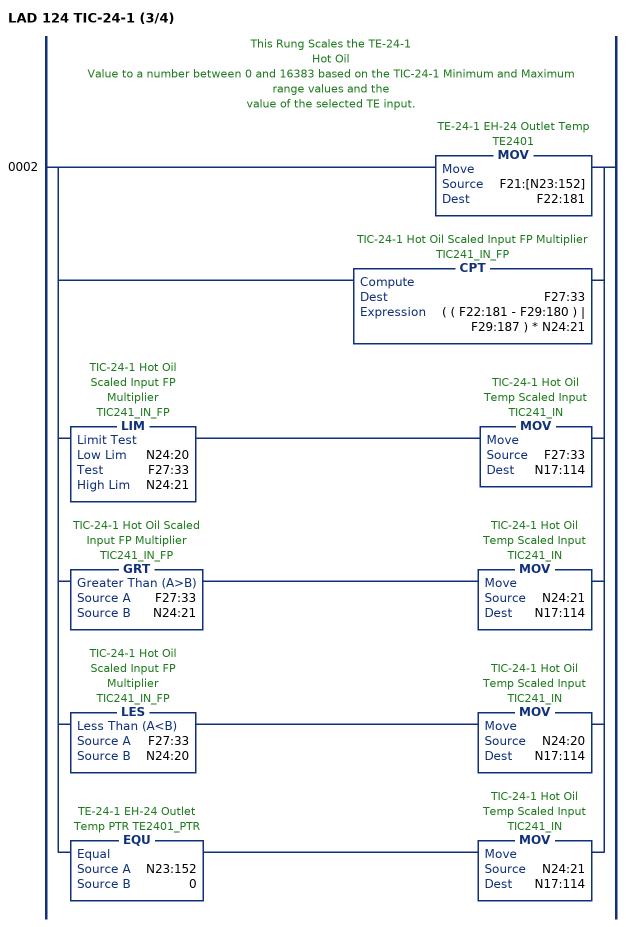
% Rung: 2 %
% This Rung Scales the TE-24-1
% Hot Oil
% Value to a number between 0 and 16383 based on the TIC-24-1 Minimum and Maximum range values and the
% value of the selected TE input. %
SOR BST MOV F21:[N23:152] F22:181 NXB CPT F27:33 " ( ( F22:181 - F29:180 ) | F29:187 ) * N24:21 " NXB LIM N24:20 F27:33 N24:21 MOV F27:33 N17:114 NXB GRT F27:33 N24:21 MOV N24:21 N17:114 NXB LES F27:33 N24:20 MOV N24:20 N17:114 NXB EQU N23:152 0 MOV N24:21 N17:114 BND EOR
%   N23:152  TE2401_PTR  "TE-24-1 EH-24 Outlet Temp PTR" %
%   F22:181  TE2401  "TE-24-1 EH-24 Outlet Temp" %
%   F27:33  TIC241_IN_FP  "TIC-24-1 Hot Oil Scaled Input FP Multiplier" %
%   F29:180  TIC241_MIN  "TIC-24-1 0% Value (For HMI Display)" %
%   F29:187  TIC241_RANGE  "TIC-24-1 Range Value (For HMI Display)" %
%   N24:21  PID_MAX  "PID Statement Maximum Value" %
%   N24:20  PID_MIN  "PID Statement Minimum Value" %
%   N17:114  TIC241_IN  "TIC-24-1 Hot Oil Temp Scaled Input" %

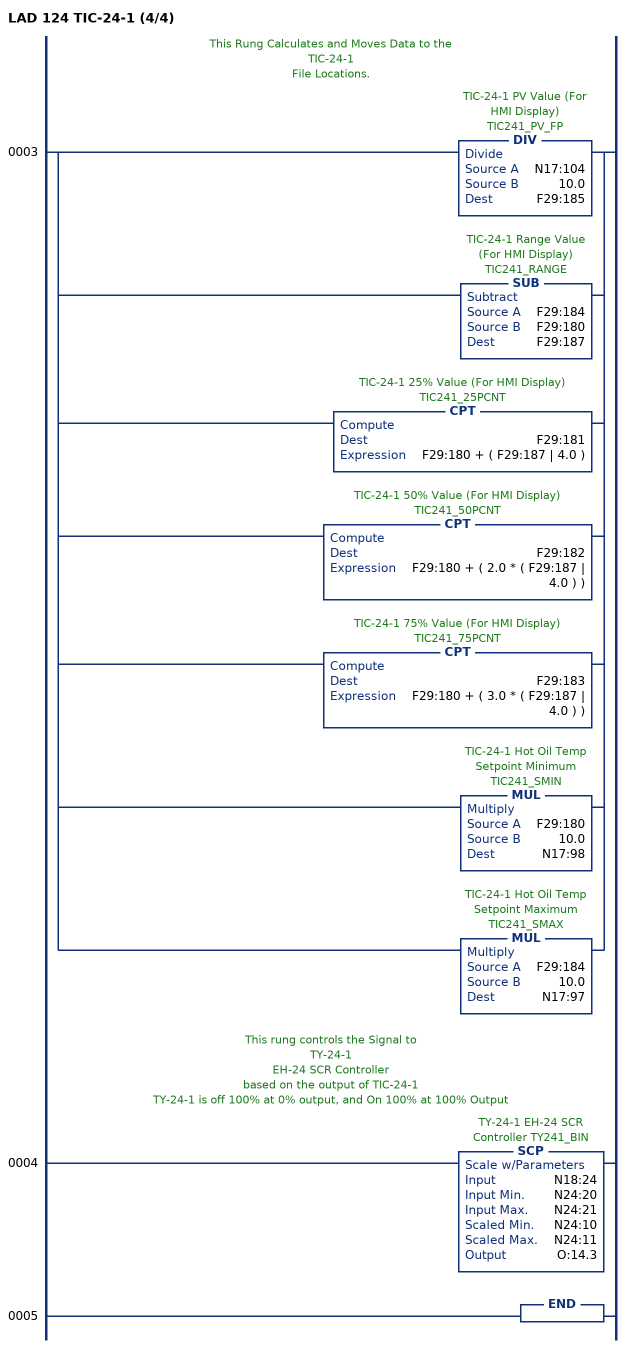
% Rung: 3 %
% This Rung Calculates and Moves Data to the
% TIC-24-1
% File Locations. %
SOR BST DIV N17:104 10.0 F29:185 NXB SUB F29:184 F29:180 F29:187 NXB CPT F29:181 " F29:180 + ( F29:187 | 4.0 ) " NXB CPT F29:182 " F29:180 + ( 2.0 * ( F29:187 | 4.0 ) ) " NXB CPT F29:183 " F29:180 + ( 3.0 * ( F29:187 | 4.0 ) ) " NXB MUL F29:180 10.0 N17:98 NXB MUL F29:184 10.0 N17:97 BND EOR
%   N17:104  TIC241_PV  "TIC-24-1 Hot Oil Temp Scaled Process Variable" %
%   F29:185  TIC241_PV_FP  "TIC-24-1 PV Value (For HMI Display)" %
%   F29:184  TIC241_MAX  "TIC-24-1 100% Value (For HMI Display)" %
%   F29:180  TIC241_MIN  "TIC-24-1 0% Value (For HMI Display)" %
%   F29:187  TIC241_RANGE  "TIC-24-1 Range Value (For HMI Display)" %
%   F29:181  TIC241_25PCNT  "TIC-24-1 25% Value (For HMI Display)" %
%   F29:182  TIC241_50PCNT  "TIC-24-1 50% Value (For HMI Display)" %
%   F29:183  TIC241_75PCNT  "TIC-24-1 75% Value (For HMI Display)" %
%   N17:98  TIC241_SMIN  "TIC-24-1 Hot Oil Temp Setpoint Minimum" %
%   N17:97  TIC241_SMAX  "TIC-24-1 Hot Oil Temp Setpoint Maximum" %
% Rung: 4 %
% This rung controls the Signal to
% TY-24-1
% EH-24 SCR Controller
% based on the output of TIC-24-1
% TY-24-1 is off 100% at 0% output, and On 100% at 100% Output %
SOR SCP N18:24 N24:20 N24:21 N24:10 N24:11 O:14.3 EOR
%   N18:24  TIC241_OUT1  "TIC-24-1 Hot Oil Temp PID Output Value" %
%   N24:20  PID_MIN  "PID Statement Minimum Value" %
%   N24:21  PID_MAX  "PID Statement Maximum Value" %
%   N24:10  AO_MIN_NO4I  "Analog Output Minimum Value Generates 4 mA DC (To NO4I AO Module)" %
%   N24:11  AO_MAX_NO4I  "Analog Output Maximum Value Generates 20 mA DC (To NO4I AO Module)" %
%   O:14.3  TY241_BIN  "TY-24-1 EH-24 SCR Controller" %
% Rung: 5 %
SOR END EOR

LADDER 125 "TIC-37-1"    % Tempered Oil Loop No-3 Temperature PID Controls %
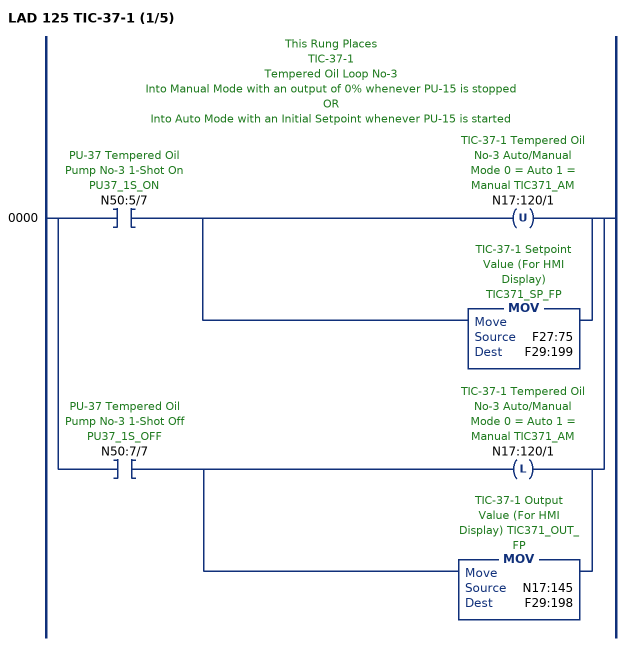
% Rung: 0 %
% This Rung Places
% TIC-37-1
% Tempered Oil Loop No-3
% Into Manual Mode with an output of 0% whenever PU-15 is stopped
% OR
% Into Auto Mode with an Initial Setpoint whenever PU-15 is started %
SOR BST XIC N50:5/7 BST OTU N17:120/1 NXB MOV F27:75 F29:199 BND NXB XIC N50:7/7 BST OTL N17:120/1 NXB MOV N17:145 F29:198 BND BND EOR
%   N50:5/7  PU37_1S_ON  "PU-37 Tempered Oil Pump No-3 1-Shot On" %
%   N17:120/1  TIC371_AM  "TIC-37-1 Tempered Oil No-3 Auto/Manual Mode 0 = Auto 1 = Manual" %
%   F27:75  TIC371_INIT_SP  "TIC-37-1 Initial Temperature Setpoint" %
%   F29:199  TIC371_SP_FP  "TIC-37-1 Setpoint Value (For HMI Display)" %
%   N50:7/7  PU37_1S_OFF  "PU-37 Tempered Oil Pump No-3 1-Shot Off" %
%   N17:145  TIC371_OFF_OUTPUT  "TIC-37-1 Output When PU-37 Is Off" %
%   F29:198  TIC371_OUT_FP  "TIC-37-1 Output Value (For HMI Display)" %

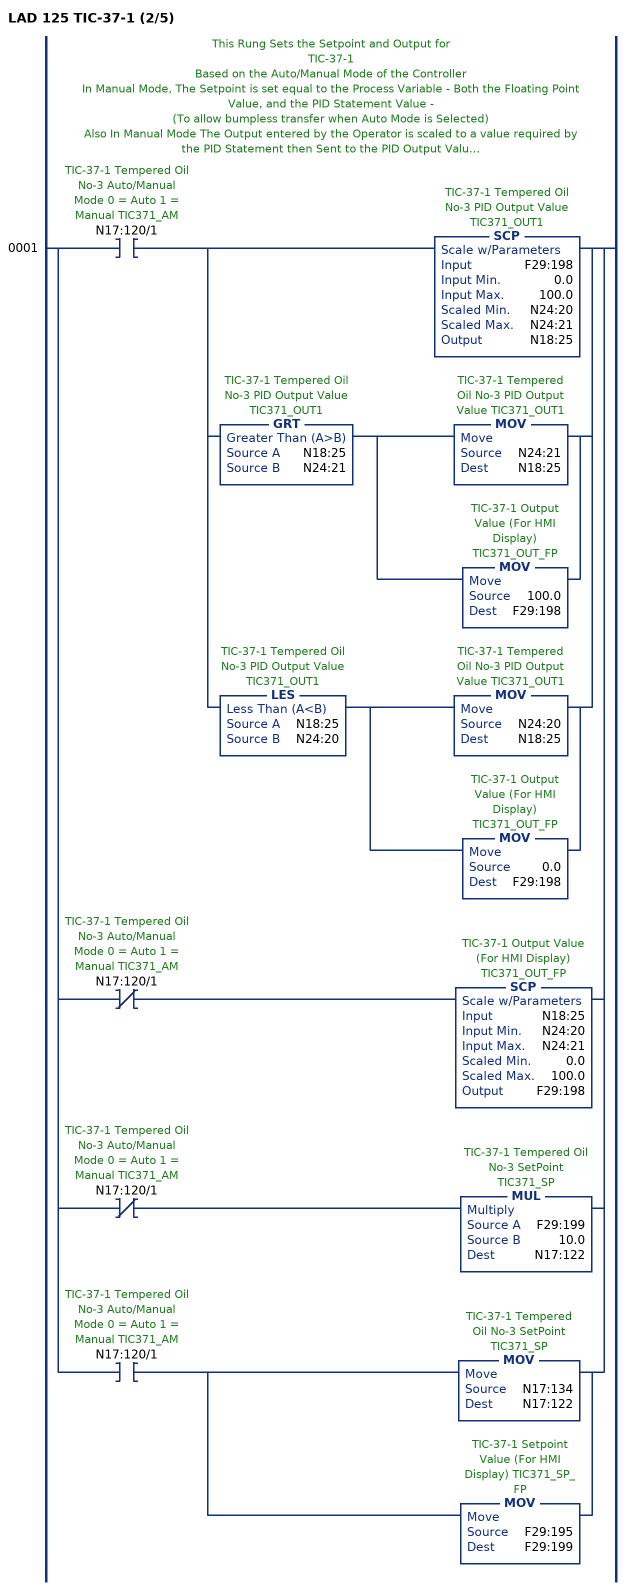
% Rung: 1 %
% This Rung Sets the Setpoint and Output for
% TIC-37-1
% Based on the Auto/Manual Mode of the Controller
% In Manual Mode, The Setpoint is set equal to the Process Variable - Both the Floating Point Value, and the PID Statement Value -
% (To allow bumpless transfer when Auto Mode is Selected)
% Also In Manual Mode The Output entered by the Operator is scaled to a value required by the PID Statement then Sent to the PID Output Value
% 
% In Auto Mode, The Setpoint is Entered by the Operator from Any HMI terminal, Multiplied by 10, and placed in the PID Statement's Setpoint Location
% Also In Auto Mode, the Output (used by the Operator) is set equal to the actual value of the pID statement
% (To allow bumpless transfer when Manual Mode is Selected) %
SOR BST XIC N17:120/1 BST SCP F29:198 0.0 100.0 N24:20 N24:21 N18:25 NXB GRT N18:25 N24:21 BST MOV N24:21 N18:25 NXB MOV 100.0 F29:198 BND NXB LES N18:25 N24:20 BST MOV N24:20 N18:25 NXB MOV 0.0 F29:198 BND BND NXB XIO N17:120/1 SCP N18:25 N24:20 N24:21 0.0 100.0 F29:198 NXB XIO N17:120/1 MUL F29:199 10.0 N17:122 NXB XIC N17:120/1 BST MOV N17:134 N17:122 NXB MOV F29:195 F29:199 BND BND EOR
%   N17:120/1  TIC371_AM  "TIC-37-1 Tempered Oil No-3 Auto/Manual Mode 0 = Auto 1 = Manual" %
%   F29:198  TIC371_OUT_FP  "TIC-37-1 Output Value (For HMI Display)" %
%   N24:20  PID_MIN  "PID Statement Minimum Value" %
%   N24:21  PID_MAX  "PID Statement Maximum Value" %
%   N18:25  TIC371_OUT1  "TIC-37-1 Tempered Oil No-3 PID Output Value" %
%   F29:199  TIC371_SP_FP  "TIC-37-1 Setpoint Value (For HMI Display)" %
%   N17:122  TIC371_SP  "TIC-37-1 Tempered Oil No-3 SetPoint" %
%   N17:134  TIC371_PV  "TIC-37-1 Tempered Oil No-3 Scaled Process Variable" %
%   F29:195  TIC371_PV_FP  "TIC-37-1 PV Value (For HMI Display)" %

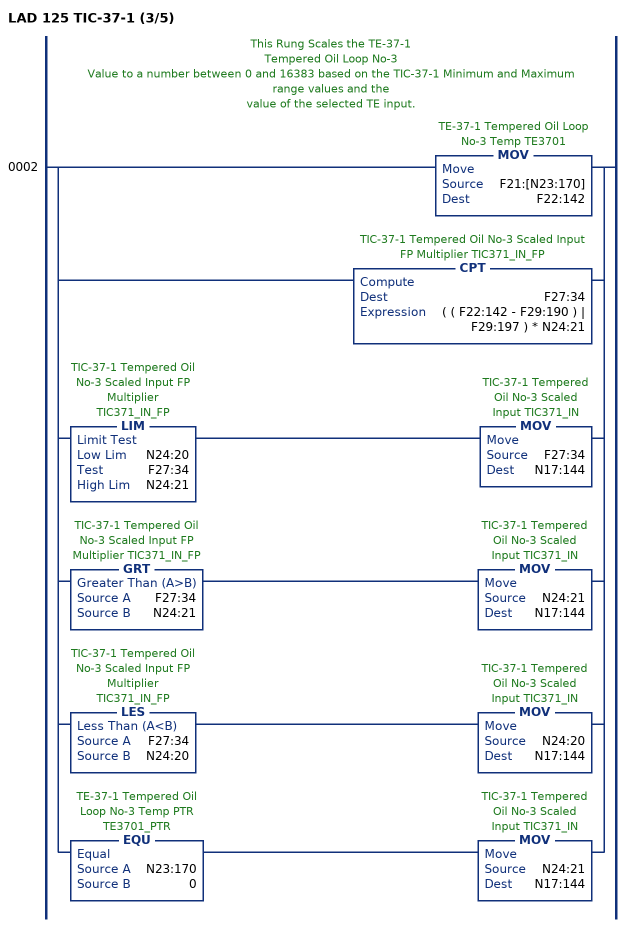
% Rung: 2 %
% This Rung Scales the TE-37-1
% Tempered Oil Loop No-3
% Value to a number between 0 and 16383 based on the TIC-37-1 Minimum and Maximum range values and the
% value of the selected TE input. %
SOR BST MOV F21:[N23:170] F22:142 NXB CPT F27:34 " ( ( F22:142 - F29:190 ) | F29:197 ) * N24:21 " NXB LIM N24:20 F27:34 N24:21 MOV F27:34 N17:144 NXB GRT F27:34 N24:21 MOV N24:21 N17:144 NXB LES F27:34 N24:20 MOV N24:20 N17:144 NXB EQU N23:170 0 MOV N24:21 N17:144 BND EOR
%   N23:170  TE3701_PTR  "TE-37-1 Tempered Oil Loop No-3 Temp PTR" %
%   F22:142  TE3701  "TE-37-1 Tempered Oil Loop No-3 Temp" %
%   F27:34  TIC371_IN_FP  "TIC-37-1 Tempered Oil No-3 Scaled Input FP Multiplier" %
%   F29:190  TIC371_MIN  "TIC-37-1 0% Value (For HMI Display)" %
%   F29:197  TIC371_RANGE  "TIC-37-1 Range Value (For HMI Display)" %
%   N24:21  PID_MAX  "PID Statement Maximum Value" %
%   N24:20  PID_MIN  "PID Statement Minimum Value" %
%   N17:144  TIC371_IN  "TIC-37-1 Tempered Oil No-3 Scaled Input" %

